FUNCTION_BLOCK Motor
VAR_INPUT
	Start: BOOL;
	Stop : BOOL;
	Overload : BOOL;
END_VAR
VAR_OUTPUT
	Coil : BOOL;
END_VAR
VAR
END_VAR

IF Start AND Stop = FALSE AND Overload = FALSE THEN
	Coil := TRUE;
ELSE
	Coil := FALSE;
	
END_IF

END_FUNCTION_BLOCK

(* stored: Version 1.1.0.1, ProductVersion 3.1.4024.9
   POU Motor: Id {9125a4ce-eef6-4d79-ade4-30c1d396401a}, SpecialFunc None *)
